{attribute 'linkalways'} 
{attribute 'no_explicit_call' := 'This FB is a CLASS and must be accessed using methods or properties'}
{attribute 'enable_dynamic_creation'}
FUNCTION_BLOCK MetadataAddedEvent EXTENDS Disposable IMPLEMENTS I_MetadataAddedEvent
VAR
	_target : I_Metadata;
END_VAR

METHOD FB_init : BOOL
VAR_INPUT
	bInitRetains : BOOL; // if TRUE, the retain variables are initialized (warm start / cold start)
	bInCopyCode : BOOL;  // if TRUE, the instance afterwards gets moved into the copy code (online change)
	Target : I_Metadata;
END_VAR
This^._target := Target;
END_METHOD

PROPERTY PUBLIC Target : I_Metadata
GET
Target := _target;
END_GET
END_PROPERTY

END_FUNCTION_BLOCK

(* stored: Version 1.1.0.1, ProductVersion 3.1.4024.12
   POU MetadataAddedEvent: Id {4b586b61-002e-0aa6-268a-625bc491caae}, SpecialFunc None
   Folder Constructor: Id {52f3fed6-5729-0c1f-250e-a1b147ab79d0}
   Method FB_init: Id {dfe44f78-6614-0ed0-1b59-7012c20527cc}
   Property Target: Id {4e432c1c-c980-0fe7-2b2e-5da9fb5af2f2}
   Get Get: Id {91df58c9-bd98-02e8-2dfc-79ec1d55dcdb} *)
